TYPE ST_MotionParameters :
STRUCT
	bClosedLoopStart : BOOL; 
	bOpenLoopStart : BOOL; 
	bWinchEnable : BOOL;
	bCylinderEnable : BOOL; 
END_STRUCT
END_TYPE

(* stored: Version 1.1.0.1, ProductVersion 3.1.4024.12
   DUT ST_MotionParameters: Id {99d50c99-7d1d-4ef9-91f7-53031211b963} *)
